LIN {X 0,Y 130.101,Z 635.486,A -85,B 0,C 180,E1 -28089.915,E2 -28089.915} C_VEL
LIN {X 0,Y 131.994,Z 639.477,A -85,B 0,C 180,E1 -28094.65,E2 -28094.65} C_VEL
LIN {X 0,Y 134.028,Z 643.617,A -85,B 0,C 180,E1 -28098.338,E2 -28098.338} C_VEL
LIN {X 0,Y 135.61,Z 647.254,A -85,B 0,C 180,E1 -28100.774,E2 -28100.774} C_VEL
LIN {X 0,Y 137.735,Z 654.472,A -85,B 0,C 180,E1 -28103.892,E2 -28103.892} C_VEL
LIN {X 0,Y 137.859,Z 654.961,A -85,B 0,C 180,E1 -28104.069,E2 -28104.069} C_VEL
LIN {X 0,Y 135.744,Z 673.421,A -85,B 0,C 180,E1 -28104.773,E2 -28104.773} C_VEL
LIN {X 0,Y 133.064,Z 685.971,A -85,B 0,C 180,E1 -28105.484,E2 -28105.484} C_VEL
LIN {X 0,Y 129.454,Z 697.536,A -85,B 0,C 180,E1 -28106.398,E2 -28106.398} C_VEL
LIN {X 0,Y 124.264,Z 710.187,A -85,B 0,C 180,E1 -28107.914,E2 -28107.914} C_VEL
LIN {X 0,Y 118.421,Z 721.436,A -85,B 0,C 180,E1 -28109.785,E2 -28109.785} C_VEL
LIN {X 0,Y 112.069,Z 731.569,A -85,B 0,C 180,E1 -28112.163,E2 -28112.163} C_VEL
LIN {X 0,Y 105.268,Z 740.708,A -85,B 0,C 180,E1 -28115.136,E2 -28115.136} C_VEL
LIN {X 0,Y 97.575,Z 749.621,A -85,B 0,C 180,E1 -28119.266,E2 -28119.266} C_VEL
LIN {X 0,Y 91.733,Z 755.687,A -85,B 0,C 180,E1 -28123.304,E2 -28123.304} C_VEL
LIN {X 0,Y 85.339,Z 761.645,A -85,B 0,C 180,E1 -28128.795,E2 -28128.795} C_VEL
LIN {X 0,Y 79.706,Z 766.355,A -85,B 0,C 180,E1 -28135.037,E2 -28135.037} C_VEL
LIN {X 0,Y 75.138,Z 769.96,A -85,B 0,C 180,E1 -28142.122,E2 -28142.122} C_VEL
LIN {X 0,Y 72.891,Z 771.823,A -85,B 0,C 180,E1 -28147.32,E2 -28147.32} C_VEL
LIN {X 0,Y 70.141,Z 774.222,A -85,B 0,C 180,E1 -28158.445,E2 -28158.445} C_VEL
LIN {X 0,Y 69.62,Z 774.834,A -85,B 0,C 180,E1 -28164.211,E2 -28164.211} C_VEL
LIN {X 0,Y 69.697,Z 775.05,A -85,B 0,C 180,E1 -28170.005,E2 -28170.005} C_VEL
LIN {X 0,Y 70.018,Z 774.825,A -85,B 0,C 180,E1 -28175.766,E2 -28175.766} C_VEL
LIN {X 0,Y 72.282,Z 773.204,A -85,B 0,C 180,E1 -28186.964,E2 -28186.964} C_VEL
LIN {X 0,Y 74.383,Z 771.8,A -85,B 0,C 180,E1 -28192.211,E2 -28192.211} C_VEL
LIN {X 0,Y 78.746,Z 768.868,A -85,B 0,C 180,E1 -28199.402,E2 -28199.402} C_VEL
LIN {X 0,Y 84.587,Z 764.915,A -85,B 0,C 180,E1 -28205.568,E2 -28205.568} C_VEL
LIN {X 0,Y 91.639,Z 759.801,A -85,B 0,C 180,E1 -28210.688,E2 -28210.688} C_VEL
LIN {X 0,Y 95.835,Z 756.939,A -85,B 0,C 180,E1 -28212.898,E2 -28212.898} C_VEL
LIN {X 0,Y 96.87,Z 757.298,A -85,B 0,C 180,E1 -28213.574,E2 -28213.574} C_VEL
LIN {X 0,Y 98.917,Z 759.037,A -85,B 0,C 180,E1 -28215.28,E2 -28215.28} C_VEL
LIN {X 0,Y 97.206,Z 757.454,A -85,B 0,C 180,E1 -28217.356,E2 -28217.356} C_VEL
LIN {X 0,Y 92.069,Z 751.92,A -85,B 0,C 180,E1 -28222.362,E2 -28222.362} C_VEL
LIN {X 0,Y 90.262,Z 751.095,A -85,B 0,C 180,E1 -28223.926,E2 -28223.926} C_VEL
LIN {X 0,Y 88.148,Z 750.795,A -85,B 0,C 180,E1 -28226.075,E2 -28226.075} C_VEL
LIN {X 0,Y 85.833,Z 749.445,A -85,B 0,C 180,E1 -28230.575,E2 -28230.575} C_VEL
LIN {X 0,Y 84.652,Z 747.487,A -85,B 0,C 180,E1 -28235.474,E2 -28235.474} C_VEL
LIN {X 0,Y 82.936,Z 746.489,A -85,B 0,C 180,E1 -28240.187,E2 -28240.187} C_VEL
LIN {X 0,Y 83.105,Z 742.849,A -85,B 0,C 180,E1 -28250.263,E2 -28250.263} C_VEL
LIN {X 0,Y 83.768,Z 741.308,A -85,B 0,C 180,E1 -28255.188,E2 -28255.188} C_VEL
LIN {X 0,Y 85.278,Z 739.422,A -85,B 0,C 180,E1 -28260,E2 -28260} C_VEL
LIN {X 0,Y 85.366,Z 739.328,A -85,B 0,C 180,E1 -28260.283,E2 -28260.283} C_VEL
LIN {X 0,Y 85.77,Z 738.947,A -85,B 0,C 180,E1 -28262.962,E2 -28262.962} C_VEL
LIN {X 0,Y 86.107,Z 739.875,A -85,B 0,C 180,E1 -28271.99,E2 -28271.99} C_VEL
LIN {X 0,Y 87.578,Z 739.192,A -85,B 0,C 180,E1 -28274.351,E2 -28274.351} C_VEL
LIN {X 0,Y 94.778,Z 735.064,A -85,B 0,C 180,E1 -28280.479,E2 -28280.479} C_VEL
LIN {X 0,Y 97.805,Z 733.364,A -85,B 0,C 180,E1 -28282.53,E2 -28282.53} C_VEL
LIN {X 0,Y 107.635,Z 727.025,A -85,B 0,C 180,E1 -28287.198,E2 -28287.198} C_VEL
LIN {X 0,Y 110.924,Z 724.845,A -85,B 0,C 180,E1 -28288.551,E2 -28288.551} C_VEL
LIN {X 0,Y 110.69,Z 725.783,A -85,B 0,C 180,E1 -28289.183,E2 -28289.183} C_VEL
LIN {X 0,Y 103.664,Z 735.37,A -85,B 0,C 180,E1 -28292.059,E2 -28292.059} C_VEL
LIN {X 0,Y 96.172,Z 744.056,A -85,B 0,C 180,E1 -28295.777,E2 -28295.777} C_VEL
LIN {X 0,Y 88.222,Z 751.991,A -85,B 0,C 180,E1 -28300.812,E2 -28300.812} C_VEL
LIN {X 0,Y 81.241,Z 757.929,A -85,B 0,C 180,E1 -28306.201,E2 -28306.201} C_VEL
LIN {X 0,Y 75.13,Z 762.615,A -85,B 0,C 180,E1 -28312.547,E2 -28312.547} C_VEL
LIN {X 0,Y 70.064,Z 766.192,A -85,B 0,C 180,E1 -28319.893,E2 -28319.893} C_VEL
LIN {X 0,Y 67.35,Z 768.037,A -85,B 0,C 180,E1 -28325.324,E2 -28325.324} C_VEL
LIN {X 0,Y 65.246,Z 769.422,A -85,B 0,C 180,E1 -28331.141,E2 -28331.141} C_VEL
LIN {X 0,Y 62.947,Z 771.009,A -85,B 0,C 180,E1 -28343.584,E2 -28343.584} C_VEL
LIN {X 0,Y 62.722,Z 771.232,A -85,B 0,C 180,E1 -28349.995,E2 -28349.995} C_VEL
LIN {X 0,Y 62.94,Z 771.037,A -85,B 0,C 180,E1 -28356.406,E2 -28356.406} C_VEL
LIN {X 0,Y 65.24,Z 769.487,A -85,B 0,C 180,E1 -28368.849,E2 -28368.849} C_VEL
LIN {X 0,Y 67.335,Z 768.13,A -85,B 0,C 180,E1 -28374.671,E2 -28374.671} C_VEL
LIN {X 0,Y 71.588,Z 765.258,A -85,B 0,C 180,E1 -28382.674,E2 -28382.674} C_VEL
LIN {X 0,Y 76.942,Z 761.361,A -85,B 0,C 180,E1 -28389.74,E2 -28389.74} C_VEL
LIN {X 0,Y 83.405,Z 756.331,A -85,B 0,C 180,E1 -28395.739,E2 -28395.739} C_VEL
LIN {X 0,Y 90.53,Z 749.996,A -85,B 0,C 180,E1 -28400.918,E2 -28400.918} C_VEL
LIN {X 0,Y 97.951,Z 742.366,A -85,B 0,C 180,E1 -28405.232,E2 -28405.232} C_VEL
LIN {X 0,Y 104.983,Z 733.989,A -85,B 0,C 180,E1 -28408.592,E2 -28408.592} C_VEL
LIN {X 0,Y 112.098,Z 724.12,A -85,B 0,C 180,E1 -28411.362,E2 -28411.362} C_VEL
LIN {X 0,Y 118.676,Z 713,A -85,B 0,C 180,E1 -28413.592,E2 -28413.592} C_VEL
LIN {X 0,Y 123.89,Z 702.094,A -85,B 0,C 180,E1 -28415.174,E2 -28415.174} C_VEL
LIN {X 0,Y 128.41,Z 690.022,A -85,B 0,C 180,E1 -28416.447,E2 -28416.447} C_VEL
LIN {X 0,Y 131.787,Z 677.536,A -85,B 0,C 180,E1 -28417.401,E2 -28417.401} C_VEL
LIN {X 0,Y 134.061,Z 664.506,A -85,B 0,C 180,E1 -28418.001,E2 -28418.001} C_VEL
LIN {X 0,Y 134.925,Z 656.287,A -85,B 0,C 180,E1 -28418.316,E2 -28418.316} C_VEL
LIN {X 0,Y 132.623,Z 650.593,A -85,B 0,C 180,E1 -28421.96,E2 -28421.96} C_VEL
LIN {X 0,Y 131.039,Z 647.12,A -85,B 0,C 180,E1 -28424.964,E2 -28424.964} C_VEL
LIN {X 0,Y 129.869,Z 644.563,A -85,B 0,C 180,E1 -28427.697,E2 -28427.697} C_VEL
LIN {X 0,Y 128.772,Z 641.834,A -85,B 0,C 180,E1 -28431.17,E2 -28431.17} C_VEL
LIN {X 0,Y 127.754,Z 638.206,A -85,B 0,C 180,E1 -28440,E2 -28440} C_VEL
LIN {X 0,Y 128.97,Z 642.374,A -85,B 0,C 180,E1 -28449.211,E2 -28449.211} C_VEL
LIN {X 0,Y 130.645,Z 646.219,A -85,B 0,C 180,E1 -28453.811,E2 -28453.811} C_VEL
LIN {X 0,Y 132.545,Z 650.383,A -85,B 0,C 180,E1 -28457.537,E2 -28457.537} C_VEL
LIN {X 0,Y 133.588,Z 653.255,A -85,B 0,C 180,E1 -28459.346,E2 -28459.346} C_VEL
LIN {X 0,Y 134.794,Z 657.852,A -85,B 0,C 180,E1 -28461.406,E2 -28461.406} C_VEL
LIN {X 0,Y 132.765,Z 674.133,A -85,B 0,C 180,E1 -28462.022,E2 -28462.022} C_VEL
LIN {X 0,Y 129.886,Z 686.836,A -85,B 0,C 180,E1 -28462.736,E2 -28462.736} C_VEL
LIN {X 0,Y 125.679,Z 699.334,A -85,B 0,C 180,E1 -28463.704,E2 -28463.704} C_VEL
LIN {X 0,Y 120.342,Z 711.571,A -85,B 0,C 180,E1 -28465.158,E2 -28465.158} C_VEL
LIN {X 0,Y 114.312,Z 722.477,A -85,B 0,C 180,E1 -28466.948,E2 -28466.948} C_VEL
LIN {X 0,Y 107.011,Z 733.323,A -85,B 0,C 180,E1 -28469.525,E2 -28469.525} C_VEL
LIN {X 0,Y 99.938,Z 742.137,A -85,B 0,C 180,E1 -28472.455,E2 -28472.455} C_VEL
LIN {X 0,Y 91.932,Z 750.729,A -85,B 0,C 180,E1 -28476.618,E2 -28476.618} C_VEL
LIN {X 0,Y 84.142,Z 757.985,A -85,B 0,C 180,E1 -28481.928,E2 -28481.928} C_VEL
LIN {X 0,Y 77.94,Z 763.129,A -85,B 0,C 180,E1 -28487.452,E2 -28487.452} C_VEL
LIN {X 0,Y 72.171,Z 767.458,A -85,B 0,C 180,E1 -28494.254,E2 -28494.254} C_VEL
LIN {X 0,Y 68.92,Z 769.755,A -85,B 0,C 180,E1 -28499.351,E2 -28499.351} C_VEL
LIN {X 0,Y 66.352,Z 771.617,A -85,B 0,C 180,E1 -28504.939,E2 -28504.939} C_VEL
LIN {X 0,Y 64.452,Z 773.016,A -85,B 0,C 180,E1 -28510.911,E2 -28510.911} C_VEL
LIN {X 0,Y 63.177,Z 774.017,A -85,B 0,C 180,E1 -28517.151,E2 -28517.151} C_VEL
LIN {X 0,Y 62.555,Z 774.629,A -85,B 0,C 180,E1 -28523.555,E2 -28523.555} C_VEL
LIN {X 0,Y 62.607,Z 774.846,A -85,B 0,C 180,E1 -28530.006,E2 -28530.006} C_VEL
LIN {X 0,Y 62.958,Z 774.62,A -85,B 0,C 180,E1 -28536.415,E2 -28536.415} C_VEL
LIN {X 0,Y 63.936,Z 774.004,A -85,B 0,C 180,E1 -28542.705,E2 -28542.705} C_VEL
LIN {X 0,Y 67.87,Z 771.594,A -85,B 0,C 180,E1 -28554.475,E2 -28554.475} C_VEL
LIN {X 0,Y 72.662,Z 768.663,A -85,B 0,C 180,E1 -28562.144,E2 -28562.144} C_VEL
LIN {X 0,Y 78.934,Z 764.71,A -85,B 0,C 180,E1 -28568.56,E2 -28568.56} C_VEL
LIN {X 0,Y 86.371,Z 759.609,A -85,B 0,C 180,E1 -28573.765,E2 -28573.765} C_VEL
LIN {X 0,Y 89.11,Z 757.647,A -85,B 0,C 180,E1 -28575.226,E2 -28575.226} C_VEL
LIN {X 0,Y 88.589,Z 756.273,A -85,B 0,C 180,E1 -28577.598,E2 -28577.598} C_VEL
LIN {X 0,Y 86.995,Z 755.555,A -85,B 0,C 180,E1 -28579.738,E2 -28579.738} C_VEL
LIN {X 0,Y 83.333,Z 754.787,A -85,B 0,C 180,E1 -28583.818,E2 -28583.818} C_VEL
LIN {X 0,Y 80.607,Z 753.671,A -85,B 0,C 180,E1 -28588.457,E2 -28588.457} C_VEL
LIN {X 0,Y 79.042,Z 752.041,A -85,B 0,C 180,E1 -28593.604,E2 -28593.604} C_VEL
LIN {X 0,Y 77.483,Z 750.845,A -85,B 0,C 180,E1 -28598.727,E2 -28598.727} C_VEL
LIN {X 0,Y 80.273,Z 743.799,A -85,B 0,C 180,E1 -28621.798,E2 -28621.798} C_VEL
LIN {X 0,Y 87.221,Z 739.406,A -85,B 0,C 180,E1 -28633.989,E2 -28633.989} C_VEL
LIN {X 0,Y 87.578,Z 739.192,A -85,B 0,C 180,E1 -28634.351,E2 -28634.351} C_VEL
LIN {X 0,Y 89.334,Z 738.402,A -85,B 0,C 180,E1 -28636.653,E2 -28636.653} C_VEL
LIN {X 0,Y 94.231,Z 737.919,A -85,B 0,C 180,E1 -28644.554,E2 -28644.554} C_VEL
LIN {X 0,Y 96.716,Z 736.808,A -85,B 0,C 180,E1 -28646.252,E2 -28646.252} C_VEL
LIN {X 0,Y 100.251,Z 734.753,A -85,B 0,C 180,E1 -28647.772,E2 -28647.772} C_VEL
LIN {X 0,Y 100.04,Z 735.616,A -85,B 0,C 180,E1 -28648.619,E2 -28648.619} C_VEL
LIN {X 0,Y 93.013,Z 743.428,A -85,B 0,C 180,E1 -28651.777,E2 -28651.777} C_VEL
LIN {X 0,Y 85.011,Z 751.089,A -85,B 0,C 180,E1 -28656.282,E2 -28656.282} C_VEL
LIN {X 0,Y 78.699,Z 756.328,A -85,B 0,C 180,E1 -28660.612,E2 -28660.612} C_VEL
LIN {X 0,Y 71.682,Z 761.409,A -85,B 0,C 180,E1 -28666.656,E2 -28666.656} C_VEL
LIN {X 0,Y 65.756,Z 765.341,A -85,B 0,C 180,E1 -28673.99,E2 -28673.99} C_VEL
LIN {X 0,Y 60.978,Z 768.243,A -85,B 0,C 180,E1 -28682.541,E2 -28682.541} C_VEL
LIN {X 0,Y 58.576,Z 769.627,A -85,B 0,C 180,E1 -28688.897,E2 -28688.897} C_VEL
LIN {X 0,Y 55.914,Z 771.214,A -85,B 0,C 180,E1 -28702.773,E2 -28702.773} C_VEL
LIN {X 0,Y 55.649,Z 771.436,A -85,B 0,C 180,E1 -28709.994,E2 -28709.994} C_VEL
LIN {X 0,Y 55.908,Z 771.241,A -85,B 0,C 180,E1 -28717.215,E2 -28717.215} C_VEL
LIN {X 0,Y 58.569,Z 769.691,A -85,B 0,C 180,E1 -28731.093,E2 -28731.093} C_VEL
LIN {X 0,Y 60.961,Z 768.334,A -85,B 0,C 180,E1 -28737.455,E2 -28737.455} C_VEL
LIN {X 0,Y 65.72,Z 765.462,A -85,B 0,C 180,E1 -28746.02,E2 -28746.02} C_VEL
LIN {X 0,Y 71.623,Z 761.565,A -85,B 0,C 180,E1 -28753.376,E2 -28753.376} C_VEL
LIN {X 0,Y 78.616,Z 756.535,A -85,B 0,C 180,E1 -28759.445,E2 -28759.445} C_VEL
LIN {X 0,Y 86.23,Z 750.198,A -85,B 0,C 180,E1 -28764.583,E2 -28764.583} C_VEL
LIN {X 0,Y 94.364,Z 742.272,A -85,B 0,C 180,E1 -28768.918,E2 -28768.918} C_VEL
LIN {X 0,Y 102.927,Z 732.412,A -85,B 0,C 180,E1 -28772.572,E2 -28772.572} C_VEL
LIN {X 0,Y 110.359,Z 722.044,A -85,B 0,C 180,E1 -28775.152,E2 -28775.152} C_VEL
LIN {X 0,Y 117.242,Z 710.355,A -85,B 0,C 180,E1 -28777.159,E2 -28777.159} C_VEL
LIN {X 0,Y 122.546,Z 698.849,A -85,B 0,C 180,E1 -28778.624,E2 -28778.624} C_VEL
LIN {X 0,Y 126.994,Z 686.168,A -85,B 0,C 180,E1 -28779.743,E2 -28779.743} C_VEL
LIN {X 0,Y 130.191,Z 673.179,A -85,B 0,C 180,E1 -28780.551,E2 -28780.551} C_VEL
LIN {X 0,Y 132.076,Z 659.981,A -85,B 0,C 180,E1 -28781.087,E2 -28781.087} C_VEL
LIN {X 0,Y 130.017,Z 654.538,A -85,B 0,C 180,E1 -28785.097,E2 -28785.097} C_VEL
LIN {X 0,Y 128.555,Z 651.086,A -85,B 0,C 180,E1 -28788.769,E2 -28788.769} C_VEL
LIN {X 0,Y 127.631,Z 648.65,A -85,B 0,C 180,E1 -28792.087,E2 -28792.087} C_VEL
LIN {X 0,Y 126.874,Z 645.374,A -85,B 0,C 180,E1 -28800,E2 -28800} C_VEL
LIN {X 0,Y 127.833,Z 649.157,A -85,B 0,C 180,E1 -28808.381,E2 -28808.381} C_VEL
LIN {X 0,Y 129.209,Z 652.691,A -85,B 0,C 180,E1 -28812.666,E2 -28812.666} C_VEL
LIN {X 0,Y 130.913,Z 656.84,A -85,B 0,C 180,E1 -28816.407,E2 -28816.407} C_VEL
LIN {X 0,Y 131.78,Z 659.784,A -85,B 0,C 180,E1 -28818.135,E2 -28818.135} C_VEL
LIN {X 0,Y 132.024,Z 660.831,A -85,B 0,C 180,E1 -28818.626,E2 -28818.626} C_VEL
LIN {X 0,Y 130.145,Z 674.683,A -85,B 0,C 180,E1 -28819.16,E2 -28819.16} C_VEL
LIN {X 0,Y 127.018,Z 687.602,A -85,B 0,C 180,E1 -28819.853,E2 -28819.853} C_VEL
LIN {X 0,Y 122.949,Z 699.261,A -85,B 0,C 180,E1 -28820.687,E2 -28820.687} C_VEL
LIN {X 0,Y 117.499,Z 711.372,A -85,B 0,C 180,E1 -28822.021,E2 -28822.021} C_VEL
LIN {X 0,Y 111.276,Z 722.276,A -85,B 0,C 180,E1 -28823.689,E2 -28823.689} C_VEL
LIN {X 0,Y 103.692,Z 733.121,A -85,B 0,C 180,E1 -28826.105,E2 -28826.105} C_VEL
LIN {X 0,Y 96.304,Z 741.934,A -85,B 0,C 180,E1 -28828.877,E2 -28828.877} C_VEL
LIN {X 0,Y 87.866,Z 750.526,A -85,B 0,C 180,E1 -28832.883,E2 -28832.883} C_VEL
LIN {X 0,Y 80.035,Z 757.41,A -85,B 0,C 180,E1 -28837.794,E2 -28837.794} C_VEL
LIN {X 0,Y 72.859,Z 762.925,A -85,B 0,C 180,E1 -28843.667,E2 -28843.667} C_VEL
LIN {X 0,Y 66.524,Z 767.254,A -85,B 0,C 180,E1 -28850.67,E2 -28850.67} C_VEL
LIN {X 0,Y 62.901,Z 769.551,A -85,B 0,C 180,E1 -28856.044,E2 -28856.044} C_VEL
LIN {X 0,Y 59.955,Z 771.412,A -85,B 0,C 180,E1 -28862.045,E2 -28862.045} C_VEL
LIN {X 0,Y 57.761,Z 772.811,A -85,B 0,C 180,E1 -28868.598,E2 -28868.598} C_VEL
LIN {X 0,Y 56.265,Z 773.812,A -85,B 0,C 180,E1 -28875.54,E2 -28875.54} C_VEL
LIN {X 0,Y 55.512,Z 774.425,A -85,B 0,C 180,E1 -28882.733,E2 -28882.733} C_VEL
LIN {X 0,Y 55.506,Z 774.641,A -85,B 0,C 180,E1 -28890.006,E2 -28890.006} C_VEL
LIN {X 0,Y 55.927,Z 774.416,A -85,B 0,C 180,E1 -28897.225,E2 -28897.225} C_VEL
LIN {X 0,Y 58.854,Z 772.794,A -85,B 0,C 180,E1 -28910.998,E2 -28910.998} C_VEL
LIN {X 0,Y 61.493,Z 771.39,A -85,B 0,C 180,E1 -28917.21,E2 -28917.21} C_VEL
LIN {X 0,Y 66.78,Z 768.458,A -85,B 0,C 180,E1 -28925.374,E2 -28925.374} C_VEL
LIN {X 0,Y 73.534,Z 764.505,A -85,B 0,C 180,E1 -28931.998,E2 -28931.998} C_VEL
LIN {X 0,Y 81.211,Z 759.537,A -85,B 0,C 180,E1 -28937.128,E2 -28937.128} C_VEL
LIN {X 0,Y 80.023,Z 758.768,A -85,B 0,C 180,E1 -28939.377,E2 -28939.377} C_VEL
LIN {X 0,Y 75.364,Z 757.491,A -85,B 0,C 180,E1 -28945.977,E2 -28945.977} C_VEL
LIN {X 0,Y 71.348,Z 752.029,A -85,B 0,C 180,E1 -28968.638,E2 -28968.638} C_VEL
LIN {X 0,Y 81.659,Z 744.392,A -85,B 0,C 180,E1 -28994.963,E2 -28994.963} C_VEL
LIN {X 0,Y 85.958,Z 742.211,A -85,B 0,C 180,E1 -28999.09,E2 -28999.09} C_VEL
LIN {X 0,Y 94.238,Z 738.135,A -85,B 0,C 180,E1 -29004.99,E2 -29004.99} C_VEL
LIN {X 0,Y 96.716,Z 736.808,A -85,B 0,C 180,E1 -29006.252,E2 -29006.252} C_VEL
LIN {X 0,Y 95.752,Z 737.763,A -85,B 0,C 180,E1 -29006.451,E2 -29006.451} C_VEL
LIN {X 0,Y 90.525,Z 741.419,A -85,B 0,C 180,E1 -29005.328,E2 -29005.328} C_VEL
LIN {X 0,Y 84.388,Z 745.051,A -85,B 0,C 180,E1 -29003.097,E2 -29003.097} C_VEL
LIN {X 0,Y 80.227,Z 747.13,A -85,B 0,C 180,E1 -29000.612,E2 -29000.612} C_VEL
LIN {X 0,Y 75.908,Z 748.925,A -85,B 0,C 180,E1 -28996.127,E2 -28996.127} C_VEL
LIN {X 0,Y 65.957,Z 754.628,A -85,B 0,C 180,E1 -28973.884,E2 -28973.884} C_VEL
LIN {X 0,Y 67.632,Z 759.85,A -85,B 0,C 180,E1 -28948.697,E2 -28948.697} C_VEL
LIN {X 0,Y 71.427,Z 761.31,A -85,B 0,C 180,E1 -28940.993,E2 -28940.993} C_VEL
LIN {X 0,Y 72.467,Z 761.915,A -85,B 0,C 180,E1 -28938.717,E2 -28938.717} C_VEL
LIN {X 0,Y 63.44,Z 767.03,A -85,B 0,C 180,E1 -28931.665,E2 -28931.665} C_VEL
LIN {X 0,Y 59.022,Z 769.319,A -85,B 0,C 180,E1 -28926.546,E2 -28926.546} C_VEL
LIN {X 0,Y 55.275,Z 771.184,A -85,B 0,C 180,E1 -28920.577,E2 -28920.577} C_VEL
LIN {X 0,Y 50.172,Z 773.594,A -85,B 0,C 180,E1 -28906.277,E2 -28906.277} C_VEL
LIN {X 0,Y 48.893,Z 774.211,A -85,B 0,C 180,E1 -28898.271,E2 -28898.271} C_VEL
LIN {X 0,Y 48.423,Z 774.437,A -85,B 0,C 180,E1 -28890.007,E2 -28890.007} C_VEL
LIN {X 0,Y 48.472,Z 774.22,A -85,B 0,C 180,E1 -28881.671,E2 -28881.671} C_VEL
LIN {X 0,Y 51.174,Z 772.605,A -85,B 0,C 180,E1 -28865.677,E2 -28865.677} C_VEL
LIN {X 0,Y 53.75,Z 771.206,A -85,B 0,C 180,E1 -28858.473,E2 -28858.473} C_VEL
LIN {X 0,Y 59.09,Z 768.271,A -85,B 0,C 180,E1 -28849.152,E2 -28849.152} C_VEL
LIN {X 0,Y 65.675,Z 764.305,A -85,B 0,C 180,E1 -28841.497,E2 -28841.497} C_VEL
LIN {X 0,Y 74.001,Z 758.608,A -85,B 0,C 180,E1 -28834.738,E2 -28834.738} C_VEL
LIN {X 0,Y 82.774,Z 751.559,A -85,B 0,C 180,E1 -28829.518,E2 -28829.518} C_VEL
LIN {X 0,Y 91.572,Z 743.304,A -85,B 0,C 180,E1 -28825.614,E2 -28825.614} C_VEL
LIN {X 0,Y 99.196,Z 734.858,A -85,B 0,C 180,E1 -28822.931,E2 -28822.931} C_VEL
LIN {X 0,Y 107.028,Z 724.426,A -85,B 0,C 180,E1 -28820.664,E2 -28820.664} C_VEL
LIN {X 0,Y 114.221,Z 712.682,A -85,B 0,C 180,E1 -28818.922,E2 -28818.922} C_VEL
LIN {X 0,Y 119.725,Z 701.262,A -85,B 0,C 180,E1 -28817.711,E2 -28817.711} C_VEL
LIN {X 0,Y 124.229,Z 689.153,A -85,B 0,C 180,E1 -28816.876,E2 -28816.876} C_VEL
LIN {X 0,Y 127.715,Z 675.876,A -85,B 0,C 180,E1 -28816.221,E2 -28816.221} C_VEL
LIN {X 0,Y 129.547,Z 664.049,A -85,B 0,C 180,E1 -28815.739,E2 -28815.739} C_VEL
LIN {X 0,Y 128.25,Z 660.288,A -85,B 0,C 180,E1 -28812.662,E2 -28812.662} C_VEL
LIN {X 0,Y 127.211,Z 657.494,A -85,B 0,C 180,E1 -28809.54,E2 -28809.54} C_VEL
LIN {X 0,Y 126.484,Z 655.285,A -85,B 0,C 180,E1 -28806.38,E2 -28806.38} C_VEL
LIN {X 0,Y 125.989,Z 652.577,A -85,B 0,C 180,E1 -28800,E2 -28800} C_VEL
LIN {X 0,Y 126.739,Z 655.984,A -85,B 0,C 180,E1 -28792.031,E2 -28792.031} C_VEL
LIN {X 0,Y 127.908,Z 659.378,A -85,B 0,C 180,E1 -28787.908,E2 -28787.908} C_VEL
LIN {X 0,Y 129.287,Z 663.248,A -85,B 0,C 180,E1 -28784.431,E2 -28784.431} C_VEL
LIN {X 0,Y 129.501,Z 663.935,A -85,B 0,C 180,E1 -28783.927,E2 -28783.927} C_VEL
LIN {X 0,Y 127.151,Z 677.322,A -85,B 0,C 180,E1 -28783.338,E2 -28783.338} C_VEL
LIN {X 0,Y 123.86,Z 689.18,A -85,B 0,C 180,E1 -28782.584,E2 -28782.584} C_VEL
LIN {X 0,Y 119.339,Z 700.928,A -85,B 0,C 180,E1 -28781.573,E2 -28781.573} C_VEL
LIN {X 0,Y 113.867,Z 711.978,A -85,B 0,C 180,E1 -28780.251,E2 -28780.251} C_VEL
LIN {X 0,Y 107.576,Z 722.245,A -85,B 0,C 180,E1 -28778.575,E2 -28778.575} C_VEL
LIN {X 0,Y 99.861,Z 732.613,A -85,B 0,C 180,E1 -28776.184,E2 -28776.184} C_VEL
LIN {X 0,Y 92.355,Z 740.997,A -85,B 0,C 180,E1 -28773.39,E2 -28773.39} C_VEL
LIN {X 0,Y 83.914,Z 749.02,A -85,B 0,C 180,E1 -28769.434,E2 -28769.434} C_VEL
LIN {X 0,Y 76.863,Z 754.757,A -85,B 0,C 180,E1 -28765.37,E2 -28765.37} C_VEL
LIN {X 0,Y 69.087,Z 760.203,A -85,B 0,C 180,E1 -28759.717,E2 -28759.717} C_VEL
LIN {X 0,Y 62.162,Z 764.467,A -85,B 0,C 180,E1 -28752.708,E2 -28752.708} C_VEL
LIN {X 0,Y 58.165,Z 766.722,A -85,B 0,C 180,E1 -28747.16,E2 -28747.16} C_VEL
LIN {X 0,Y 54.743,Z 768.539,A -85,B 0,C 180,E1 -28740.891,E2 -28740.891} C_VEL
LIN {X 0,Y 50.037,Z 770.861,A -85,B 0,C 180,E1 -28726.307,E2 -28726.307} C_VEL
LIN {X 0,Y 48.874,Z 771.445,A -85,B 0,C 180,E1 -28718.261,E2 -28718.261} C_VEL
LIN {X 0,Y 48.565,Z 771.64,A -85,B 0,C 180,E1 -28709.993,E2 -28709.993} C_VEL
LIN {X 0,Y 48.878,Z 771.418,A -85,B 0,C 180,E1 -28701.726,E2 -28701.726} C_VEL
LIN {X 0,Y 50.04,Z 770.816,A -85,B 0,C 180,E1 -28693.679,E2 -28693.679} C_VEL
LIN {X 0,Y 54.761,Z 768.448,A -85,B 0,C 180,E1 -28679.105,E2 -28679.105} C_VEL
LIN {X 0,Y 60.158,Z 765.547,A -85,B 0,C 180,E1 -28670.011,E2 -28670.011} C_VEL
LIN {X 0,Y 66.696,Z 761.615,A -85,B 0,C 180,E1 -28662.464,E2 -28662.464} C_VEL
LIN {X 0,Y 74.275,Z 756.534,A -85,B 0,C 180,E1 -28656.452,E2 -28656.452} C_VEL
LIN {X 0,Y 82.373,Z 750.135,A -85,B 0,C 180,E1 -28651.432,E2 -28651.432} C_VEL
LIN {X 0,Y 88.024,Z 745.015,A -85,B 0,C 180,E1 -28648.559,E2 -28648.559} C_VEL
LIN {X 0,Y 89.392,Z 743.169,A -85,B 0,C 180,E1 -28646.973,E2 -28646.973} C_VEL
LIN {X 0,Y 80.227,Z 747.13,A -85,B 0,C 180,E1 -28640.612,E2 -28640.612} C_VEL
LIN {X 0,Y 74.947,Z 749.727,A -85,B 0,C 180,E1 -28636.69,E2 -28636.69} C_VEL
LIN {X 0,Y 64.868,Z 754.966,A -85,B 0,C 180,E1 -28627.631,E2 -28627.631} C_VEL
LIN {X 0,Y 62.176,Z 756.388,A -85,B 0,C 180,E1 -28623.108,E2 -28623.108} C_VEL
LIN {X 0,Y 61.539,Z 756.762,A -85,B 0,C 180,E1 -28621.431,E2 -28621.431} C_VEL
LIN {X 0,Y 60.042,Z 761.988,A -85,B 0,C 180,E1 -28592.082,E2 -28592.082} C_VEL
LIN {X 0,Y 62.054,Z 763.068,A -85,B 0,C 180,E1 -28585.509,E2 -28585.509} C_VEL
LIN {X 0,Y 63.705,Z 764.094,A -85,B 0,C 180,E1 -28580.564,E2 -28580.564} C_VEL
LIN {X 0,Y 55.821,Z 768.048,A -85,B 0,C 180,E1 -28573.834,E2 -28573.834} C_VEL
LIN {X 0,Y 49.303,Z 770.979,A -85,B 0,C 180,E1 -28564.772,E2 -28564.772} C_VEL
LIN {X 0,Y 43.412,Z 773.389,A -85,B 0,C 180,E1 -28548.9,E2 -28548.9} C_VEL
LIN {X 0,Y 41.897,Z 774.006,A -85,B 0,C 180,E1 -28539.665,E2 -28539.665} C_VEL
LIN {X 0,Y 41.323,Z 774.232,A -85,B 0,C 180,E1 -28530.008,E2 -28530.008} C_VEL
LIN {X 0,Y 41.446,Z 774.015,A -85,B 0,C 180,E1 -28520.246,E2 -28520.246} C_VEL
LIN {X 0,Y 44.766,Z 772.4,A -85,B 0,C 180,E1 -28501.911,E2 -28501.911} C_VEL
LIN {X 0,Y 47.81,Z 771.001,A -85,B 0,C 180,E1 -28493.994,E2 -28493.994} C_VEL
LIN {X 0,Y 53.898,Z 768.067,A -85,B 0,C 180,E1 -28484.189,E2 -28484.189} C_VEL
LIN {X 0,Y 61.195,Z 764.102,A -85,B 0,C 180,E1 -28476.504,E2 -28476.504} C_VEL
LIN {X 0,Y 69.482,Z 758.893,A -85,B 0,C 180,E1 -28470.381,E2 -28470.381} C_VEL
LIN {X 0,Y 78.01,Z 752.593,A -85,B 0,C 180,E1 -28465.733,E2 -28465.733} C_VEL
LIN {X 0,Y 87.161,Z 744.591,A -85,B 0,C 180,E1 -28461.998,E2 -28461.998} C_VEL
LIN {X 0,Y 96.646,Z 734.656,A -85,B 0,C 180,E1 -28459.043,E2 -28459.043} C_VEL
LIN {X 0,Y 104.734,Z 724.225,A -85,B 0,C 180,E1 -28457.029,E2 -28457.029} C_VEL
LIN {X 0,Y 112.123,Z 712.482,A -85,B 0,C 180,E1 -28455.493,E2 -28455.493} C_VEL
LIN {X 0,Y 117.634,Z 701.359,A -85,B 0,C 180,E1 -28454.437,E2 -28454.437} C_VEL
LIN {X 0,Y 122.227,Z 689.37,A -85,B 0,C 180,E1 -28453.719,E2 -28453.719} C_VEL
LIN {X 0,Y 125.731,Z 676.524,A -85,B 0,C 180,E1 -28453.16,E2 -28453.16} C_VEL
LIN {X 0,Y 127.22,Z 668.095,A -85,B 0,C 180,E1 -28452.766,E2 -28452.766} C_VEL
LIN {X 0,Y 126.08,Z 664.34,A -85,B 0,C 180,E1 -28448.818,E2 -28448.818} C_VEL
LIN {X 0,Y 125.463,Z 662.101,A -85,B 0,C 180,E1 -28445.626,E2 -28445.626} C_VEL
LIN {X 0,Y 125.115,Z 659.699,A -85,B 0,C 180,E1 -28440,E2 -28440} C_VEL
LIN {X 0,Y 125.671,Z 662.859,A -85,B 0,C 180,E1 -28432.771,E2 -28432.771} C_VEL
LIN {X 0,Y 126.577,Z 666.11,A -85,B 0,C 180,E1 -28428.794,E2 -28428.794} C_VEL
LIN {X 0,Y 127.166,Z 668.141,A -85,B 0,C 180,E1 -28426.839,E2 -28426.839} C_VEL
LIN {X 0,Y 124.226,Z 681.703,A -85,B 0,C 180,E1 -28426.241,E2 -28426.241} C_VEL
LIN {X 0,Y 120.593,Z 693.091,A -85,B 0,C 180,E1 -28425.49,E2 -28425.49} C_VEL
LIN {X 0,Y 115.764,Z 704.452,A -85,B 0,C 180,E1 -28424.516,E2 -28424.516} C_VEL
LIN {X 0,Y 109.245,Z 716.295,A -85,B 0,C 180,E1 -28423.114,E2 -28423.114} C_VEL
LIN {X 0,Y 101.986,Z 726.856,A -85,B 0,C 180,E1 -28421.345,E2 -28421.345} C_VEL
LIN {X 0,Y 94.062,Z 736.369,A -85,B 0,C 180,E1 -28419.049,E2 -28419.049} C_VEL
LIN {X 0,Y 84.825,Z 745.508,A -85,B 0,C 180,E1 -28415.686,E2 -28415.686} C_VEL
LIN {X 0,Y 75.926,Z 752.852,A -85,B 0,C 180,E1 -28411.554,E2 -28411.554} C_VEL
LIN {X 0,Y 67.432,Z 758.74,A -85,B 0,C 180,E1 -28406.479,E2 -28406.479} C_VEL
LIN {X 0,Y 59.559,Z 763.386,A -85,B 0,C 180,E1 -28400.076,E2 -28400.076} C_VEL
LIN {X 0,Y 52.685,Z 766.925,A -85,B 0,C 180,E1 -28391.826,E2 -28391.826} C_VEL
LIN {X 0,Y 48.78,Z 768.743,A -85,B 0,C 180,E1 -28385.182,E2 -28385.182} C_VEL
LIN {X 0,Y 43.272,Z 771.065,A -85,B 0,C 180,E1 -28368.947,E2 -28368.947} C_VEL
LIN {X 0,Y 41.877,Z 771.649,A -85,B 0,C 180,E1 -28359.653,E2 -28359.653} C_VEL
LIN {X 0,Y 41.469,Z 771.845,A -85,B 0,C 180,E1 -28349.992,E2 -28349.992} C_VEL
LIN {X 0,Y 41.881,Z 771.623,A -85,B 0,C 180,E1 -28340.331,E2 -28340.331} C_VEL
LIN {X 0,Y 43.276,Z 771.021,A -85,B 0,C 180,E1 -28331.038,E2 -28331.038} C_VEL
LIN {X 0,Y 48.799,Z 768.654,A -85,B 0,C 180,E1 -28314.816,E2 -28314.816} C_VEL
LIN {X 0,Y 54.909,Z 765.753,A -85,B 0,C 180,E1 -28305.246,E2 -28305.246} C_VEL
LIN {X 0,Y 62.125,Z 761.82,A -85,B 0,C 180,E1 -28297.629,E2 -28297.629} C_VEL
LIN {X 0,Y 70.29,Z 756.74,A -85,B 0,C 180,E1 -28291.793,E2 -28291.793} C_VEL
LIN {X 0,Y 78.896,Z 750.342,A -85,B 0,C 180,E1 -28287.018,E2 -28287.018} C_VEL
LIN {X 0,Y 79.584,Z 749.578,A -85,B 0,C 180,E1 -28286.203,E2 -28286.203} C_VEL
LIN {X 0,Y 74.338,Z 751.551,A -85,B 0,C 180,E1 -28282.22,E2 -28282.22} C_VEL
LIN {X 0,Y 66.405,Z 754.444,A -85,B 0,C 180,E1 -28272.221,E2 -28272.221} C_VEL
LIN {X 0,Y 61.539,Z 756.762,A -85,B 0,C 180,E1 -28261.431,E2 -28261.431} C_VEL
LIN {X 0,Y 59.506,Z 758.118,A -85,B 0,C 180,E1 -28256.326,E2 -28256.326} C_VEL
LIN {X 0,Y 55.587,Z 760.943,A -85,B 0,C 180,E1 -28247.669,E2 -28247.669} C_VEL
LIN {X 0,Y 53.092,Z 763.498,A -85,B 0,C 180,E1 -28237.93,E2 -28237.93} C_VEL
LIN {X 0,Y 53.408,Z 764.536,A -85,B 0,C 180,E1 -28231.706,E2 -28231.706} C_VEL
LIN {X 0,Y 54.898,Z 765.293,A -85,B 0,C 180,E1 -28226.049,E2 -28226.049} C_VEL
LIN {X 0,Y 55.039,Z 766.026,A -85,B 0,C 180,E1 -28222.828,E2 -28222.828} C_VEL
LIN {X 0,Y 48.366,Z 768.909,A -85,B 0,C 180,E1 -28216.607,E2 -28216.607} C_VEL
LIN {X 0,Y 43.673,Z 770.774,A -85,B 0,C 180,E1 -28210.078,E2 -28210.078} C_VEL
LIN {X 0,Y 36.787,Z 773.184,A -85,B 0,C 180,E1 -28192.473,E2 -28192.473} C_VEL
LIN {X 0,Y 34.929,Z 773.802,A -85,B 0,C 180,E1 -28181.618,E2 -28181.618} C_VEL
LIN {X 0,Y 34.237,Z 774.028,A -85,B 0,C 180,E1 -28170.01,E2 -28170.01} C_VEL
LIN {X 0,Y 34.467,Z 773.81,A -85,B 0,C 180,E1 -28158.245,E2 -28158.245} C_VEL
LIN {X 0,Y 38.622,Z 772.195,A -85,B 0,C 180,E1 -28136.925,E2 -28136.925} C_VEL
LIN {X 0,Y 42.245,Z 770.796,A -85,B 0,C 180,E1 -28128.294,E2 -28128.294} C_VEL
LIN {X 0,Y 49.196,Z 767.862,A -85,B 0,C 180,E1 -28118.226,E2 -28118.226} C_VEL
LIN {X 0,Y 57.252,Z 763.898,A -85,B 0,C 180,E1 -28110.776,E2 -28110.776} C_VEL
LIN {X 0,Y 66.413,Z 758.536,A -85,B 0,C 180,E1 -28104.934,E2 -28104.934} C_VEL
LIN {X 0,Y 76.762,Z 751.152,A -85,B 0,C 180,E1 -28100.222,E2 -28100.222} C_VEL
LIN {X 0,Y 86.379,Z 742.899,A -85,B 0,C 180,E1 -28097.073,E2 -28097.073} C_VEL
LIN {X 0,Y 94.563,Z 734.453,A -85,B 0,C 180,E1 -28094.962,E2 -28094.962} C_VEL
LIN {X 0,Y 102.882,Z 724.025,A -85,B 0,C 180,E1 -28093.253,E2 -28093.253} C_VEL
LIN {X 0,Y 110.441,Z 712.283,A -85,B 0,C 180,E1 -28091.948,E2 -28091.948} C_VEL
LIN {X 0,Y 116.583,Z 699.964,A -85,B 0,C 180,E1 -28090.98,E2 -28090.98} C_VEL
LIN {X 0,Y 121.448,Z 687.012,A -85,B 0,C 180,E1 -28090.357,E2 -28090.357} C_VEL
LIN {X 0,Y 124.711,Z 674.513,A -85,B 0,C 180,E1 -28089.898,E2 -28089.898} C_VEL
LIN {X 0,Y 125.046,Z 672.664,A -85,B 0,C 180,E1 -28089.819,E2 -28089.819} C_VEL
LIN {X 0,Y 124.402,Z 669.185,A -85,B 0,C 180,E1 -28085.47,E2 -28085.47} C_VEL
LIN {X 0,Y 124.144,Z 666.888,A -85,B 0,C 180,E1 -28080,E2 -28080} C_VEL
LIN {X 0,Y 124.403,Z 669.681,A -85,B 0,C 180,E1 -28073.512,E2 -28073.512} C_VEL
LIN {X 0,Y 124.94,Z 672.55,A -85,B 0,C 180,E1 -28069.924,E2 -28069.924} C_VEL
LIN {X 0,Y 122.297,Z 683.479,A -85,B 0,C 180,E1 -28069.384,E2 -28069.384} C_VEL
LIN {X 0,Y 118.015,Z 695.853,A -85,B 0,C 180,E1 -28068.643,E2 -28068.643} C_VEL
LIN {X 0,Y 113.239,Z 706.297,A -85,B 0,C 180,E1 -28067.806,E2 -28067.806} C_VEL
LIN {X 0,Y 106.573,Z 717.783,A -85,B 0,C 180,E1 -28066.565,E2 -28066.565} C_VEL
LIN {X 0,Y 99.122,Z 728.123,A -85,B 0,C 180,E1 -28065.012,E2 -28065.012} C_VEL
LIN {X 0,Y 91.766,Z 736.571,A -85,B 0,C 180,E1 -28063.186,E2 -28063.186} C_VEL
LIN {X 0,Y 82.158,Z 745.711,A -85,B 0,C 180,E1 -28060.202,E2 -28060.202} C_VEL
LIN {X 0,Y 72.804,Z 753.056,A -85,B 0,C 180,E1 -28056.488,E2 -28056.488} C_VEL
LIN {X 0,Y 63.79,Z 758.943,A -85,B 0,C 180,E1 -28051.798,E2 -28051.798} C_VEL
LIN {X 0,Y 55.273,Z 763.589,A -85,B 0,C 180,E1 -28045.727,E2 -28045.727} C_VEL
LIN {X 0,Y 47.636,Z 767.129,A -85,B 0,C 180,E1 -28037.522,E2 -28037.522} C_VEL
LIN {X 0,Y 43.172,Z 768.947,A -85,B 0,C 180,E1 -28030.619,E2 -28030.619} C_VEL
LIN {X 0,Y 36.624,Z 771.27,A -85,B 0,C 180,E1 -28012.558,E2 -28012.558} C_VEL
LIN {X 0,Y 34.894,Z 771.854,A -85,B 0,C 180,E1 -28001.609,E2 -28001.609} C_VEL
LIN {X 0,Y 34.391,Z 772.049,A -85,B 0,C 180,E1 -27989.99,E2 -27989.99} C_VEL
LIN {X 0,Y 34.898,Z 771.828,A -85,B 0,C 180,E1 -27978.372,E2 -27978.372} C_VEL
LIN {X 0,Y 39.454,Z 770.242,A -85,B 0,C 180,E1 -27957.687,E2 -27957.687} C_VEL
LIN {X 0,Y 43.191,Z 768.859,A -85,B 0,C 180,E1 -27949.382,E2 -27949.382} C_VEL
LIN {X 0,Y 50.119,Z 765.958,A -85,B 0,C 180,E1 -27939.524,E2 -27939.524} C_VEL
LIN {X 0,Y 58.067,Z 762.026,A -85,B 0,C 180,E1 -27932.078,E2 -27932.078} C_VEL
LIN {X 0,Y 66.454,Z 757.176,A -85,B 0,C 180,E1 -27926.814,E2 -27926.814} C_VEL
LIN {X 0,Y 68.428,Z 755.492,A -85,B 0,C 180,E1 -27924.257,E2 -27924.257} C_VEL
LIN {X 0,Y 52.813,Z 761.703,A -85,B 0,C 180,E1 -27892.353,E2 -27892.353} C_VEL
LIN {X 0,Y 53.408,Z 764.536,A -85,B 0,C 180,E1 -27871.706,E2 -27871.706} C_VEL
LIN {X 0,Y 53.146,Z 765.119,A -85,B 0,C 180,E1 -27869.336,E2 -27869.336} C_VEL
LIN {X 0,Y 51.503,Z 766.167,A -85,B 0,C 180,E1 -27866.765,E2 -27866.765} C_VEL
LIN {X 0,Y 47.991,Z 767.669,A -85,B 0,C 180,E1 -27863.869,E2 -27863.869} C_VEL
LIN {X 0,Y 39.894,Z 770.184,A -85,B 0,C 180,E1 -27858.291,E2 -27858.291} C_VEL
LIN {X 0,Y 37.552,Z 770.85,A -85,B 0,C 180,E1 -27855.349,E2 -27855.349} C_VEL
LIN {X 0,Y 30.355,Z 772.98,A -85,B 0,C 180,E1 -27837.597,E2 -27837.597} C_VEL
LIN {X 0,Y 28.011,Z 773.597,A -85,B 0,C 180,E1 -27824.544,E2 -27824.544} C_VEL
LIN {X 0,Y 27.123,Z 773.823,A -85,B 0,C 180,E1 -27810.013,E2 -27810.013} C_VEL
LIN {X 0,Y 27.537,Z 773.605,A -85,B 0,C 180,E1 -27795.226,E2 -27795.226} C_VEL
LIN {X 0,Y 32.885,Z 771.99,A -85,B 0,C 180,E1 -27770.137,E2 -27770.137} C_VEL
LIN {X 0,Y 37.222,Z 770.591,A -85,B 0,C 180,E1 -27760.968,E2 -27760.968} C_VEL
LIN {X 0,Y 45.135,Z 767.657,A -85,B 0,C 180,E1 -27751.099,E2 -27751.099} C_VEL
LIN {X 0,Y 53.96,Z 763.694,A -85,B 0,C 180,E1 -27744.273,E2 -27744.273} C_VEL
LIN {X 0,Y 63.342,Z 758.57,A -85,B 0,C 180,E1 -27739.297,E2 -27739.297} C_VEL
LIN {X 0,Y 72.955,Z 752.185,A -85,B 0,C 180,E1 -27735.584,E2 -27735.584} C_VEL
LIN {X 0,Y 82.893,Z 744.186,A -85,B 0,C 180,E1 -27732.855,E2 -27732.855} C_VEL
LIN {X 0,Y 92.981,Z 734.251,A -85,B 0,C 180,E1 -27730.722,E2 -27730.722} C_VEL
LIN {X 0,Y 101.489,Z 723.824,A -85,B 0,C 180,E1 -27729.346,E2 -27729.346} C_VEL
LIN {X 0,Y 109.194,Z 712.083,A -85,B 0,C 180,E1 -27728.307,E2 -27728.307} C_VEL
LIN {X 0,Y 115.216,Z 700.289,A -85,B 0,C 180,E1 -27727.548,E2 -27727.548} C_VEL
LIN {X 0,Y 120.376,Z 686.816,A -85,B 0,C 180,E1 -27727.037,E2 -27727.037} C_VEL
LIN {X 0,Y 122.972,Z 677.344,A -85,B 0,C 180,E1 -27726.676,E2 -27726.676} C_VEL
LIN {X 0,Y 122.791,Z 675.512,A -85,B 0,C 180,E1 -27723.692,E2 -27723.692} C_VEL
LIN {X 0,Y 122.837,Z 674.015,A -85,B 0,C 180,E1 -27720,E2 -27720} C_VEL
LIN {X 0,Y 122.801,Z 676.432,A -85,B 0,C 180,E1 -27714.252,E2 -27714.252} C_VEL
LIN {X 0,Y 122.869,Z 677.362,A -85,B 0,C 180,E1 -27712.96,E2 -27712.96} C_VEL
LIN {X 0,Y 119.078,Z 690.212,A -85,B 0,C 180,E1 -27712.358,E2 -27712.358} C_VEL
LIN {X 0,Y 114.215,Z 701.93,A -85,B 0,C 180,E1 -27711.695,E2 -27711.695} C_VEL
LIN {X 0,Y 108.545,Z 712.578,A -85,B 0,C 180,E1 -27710.871,E2 -27710.871} C_VEL
LIN {X 0,Y 100.904,Z 724.017,A -85,B 0,C 180,E1 -27709.654,E2 -27709.654} C_VEL
LIN {X 0,Y 93.319,Z 733.218,A -85,B 0,C 180,E1 -27708.23,E2 -27708.23} C_VEL
LIN {X 0,Y 84.976,Z 741.604,A -85,B 0,C 180,E1 -27706.338,E2 -27706.338} C_VEL
LIN {X 0,Y 75.557,Z 749.475,A -85,B 0,C 180,E1 -27703.571,E2 -27703.571} C_VEL
LIN {X 0,Y 67.083,Z 755.367,A -85,B 0,C 180,E1 -27700.526,E2 -27700.526} C_VEL
LIN {X 0,Y 57.658,Z 760.813,A -85,B 0,C 180,E1 -27696.075,E2 -27696.075} C_VEL
LIN {X 0,Y 48.674,Z 765.08,A -85,B 0,C 180,E1 -27690.02,E2 -27690.02} C_VEL
LIN {X 0,Y 43.153,Z 767.333,A -85,B 0,C 180,E1 -27684.505,E2 -27684.505} C_VEL
LIN {X 0,Y 38.07,Z 769.151,A -85,B 0,C 180,E1 -27677.584,E2 -27677.584} C_VEL
LIN {X 0,Y 30.197,Z 771.474,A -85,B 0,C 180,E1 -27657.728,E2 -27657.728} C_VEL
LIN {X 0,Y 27.971,Z 772.058,A -85,B 0,C 180,E1 -27644.539,E2 -27644.539} C_VEL
LIN {X 0,Y 27.295,Z 772.254,A -85,B 0,C 180,E1 -27629.987,E2 -27629.987} C_VEL
LIN {X 0,Y 27.976,Z 772.033,A -85,B 0,C 180,E1 -27615.438,E2 -27615.438} C_VEL
LIN {X 0,Y 30.203,Z 771.431,A -85,B 0,C 180,E1 -27602.252,E2 -27602.252} C_VEL
LIN {X 0,Y 38.089,Z 769.065,A -85,B 0,C 180,E1 -27582.42,E2 -27582.42} C_VEL
LIN {X 0,Y 45.915,Z 766.164,A -85,B 0,C 180,E1 -27572.651,E2 -27572.651} C_VEL
LIN {X 0,Y 56.596,Z 761.223,A -85,B 0,C 180,E1 -27564.614,E2 -27564.614} C_VEL
LIN {X 0,Y 58.488,Z 760.064,A -85,B 0,C 180,E1 -27562.443,E2 -27562.443} C_VEL
LIN {X 0,Y 45.561,Z 765.653,A -85,B 0,C 180,E1 -27522.031,E2 -27522.031} C_VEL
LIN {X 0,Y 46.343,Z 766.621,A -85,B 0,C 180,E1 -27512.703,E2 -27512.703} C_VEL
LIN {X 0,Y 46.285,Z 767.774,A -85,B 0,C 180,E1 -27505.655,E2 -27505.655} C_VEL
LIN {X 0,Y 37.552,Z 770.85,A -85,B 0,C 180,E1 -27495.349,E2 -27495.349} C_VEL
LIN {X 0,Y 33.339,Z 771.99,A -85,B 0,C 180,E1 -27488.843,E2 -27488.843} C_VEL
LIN {X 0,Y 26.091,Z 773.183,A -85,B 0,C 180,E1 -27475.875,E2 -27475.875} C_VEL
LIN {X 0,Y 21.471,Z 773.568,A -85,B 0,C 180,E1 -27460.055,E2 -27460.055} C_VEL
LIN {X 0,Y 20.041,Z 773.578,A -85,B 0,C 180,E1 -27443.991,E2 -27443.991} C_VEL
LIN {X 0,Y 20.144,Z 773.492,A -85,B 0,C 180,E1 -27438.324,E2 -27438.324} C_VEL
LIN {X 0,Y 23.507,Z 772.786,A -85,B 0,C 180,E1 -27413.295,E2 -27413.295} C_VEL
LIN {X 0,Y 27.787,Z 771.785,A -85,B 0,C 180,E1 -27400.663,E2 -27400.663} C_VEL
LIN {X 0,Y 32.987,Z 770.386,A -85,B 0,C 180,E1 -27391.568,E2 -27391.568} C_VEL
LIN {X 0,Y 41.9,Z 767.453,A -85,B 0,C 180,E1 -27382.724,E2 -27382.724} C_VEL
LIN {X 0,Y 51.445,Z 763.49,A -85,B 0,C 180,E1 -27377.03,E2 -27377.03} C_VEL
LIN {X 0,Y 62.978,Z 757.404,A -85,B 0,C 180,E1 -27372.492,E2 -27372.492} C_VEL
LIN {X 0,Y 73.069,Z 750.745,A -85,B 0,C 180,E1 -27369.672,E2 -27369.672} C_VEL
LIN {X 0,Y 83.317,Z 742.493,A -85,B 0,C 180,E1 -27367.668,E2 -27367.668} C_VEL
LIN {X 0,Y 91.923,Z 734.049,A -85,B 0,C 180,E1 -27366.362,E2 -27366.362} C_VEL
LIN {X 0,Y 100.581,Z 723.623,A -85,B 0,C 180,E1 -27365.355,E2 -27365.355} C_VEL
LIN {X 0,Y 108.397,Z 711.883,A -85,B 0,C 180,E1 -27364.598,E2 -27364.598} C_VEL
LIN {X 0,Y 114.196,Z 700.784,A -85,B 0,C 180,E1 -27364.052,E2 -27364.052} C_VEL
LIN {X 0,Y 119.239,Z 688.034,A -85,B 0,C 180,E1 -27363.69,E2 -27363.69} C_VEL
LIN {X 0,Y 120.985,Z 682.385,A -85,B 0,C 180,E1 -27363.517,E2 -27363.517} C_VEL
LIN {X 0,Y 121.088,Z 681.034,A -85,B 0,C 180,E1 -27360,E2 -27360} C_VEL
LIN {X 0,Y 120.896,Z 682.437,A -85,B 0,C 180,E1 -27356.112,E2 -27356.112} C_VEL
LIN {X 0,Y 116.608,Z 694.931,A -85,B 0,C 180,E1 -27355.578,E2 -27355.578} C_VEL
LIN {X 0,Y 111.111,Z 706.695,A -85,B 0,C 180,E1 -27354.973,E2 -27354.973} C_VEL
LIN {X 0,Y 104.194,Z 718.184,A -85,B 0,C 180,E1 -27354.174,E2 -27354.174} C_VEL
LIN {X 0,Y 96.429,Z 728.526,A -85,B 0,C 180,E1 -27353.194,E2 -27353.194} C_VEL
LIN {X 0,Y 88.708,Z 736.974,A -85,B 0,C 180,E1 -27351.992,E2 -27351.992} C_VEL
LIN {X 0,Y 78.489,Z 746.117,A -85,B 0,C 180,E1 -27350.019,E2 -27350.019} C_VEL
LIN {X 0,Y 68.39,Z 753.461,A -85,B 0,C 180,E1 -27347.464,E2 -27347.464} C_VEL
LIN {X 0,Y 58.442,Z 759.349,A -85,B 0,C 180,E1 -27344.141,E2 -27344.141} C_VEL
LIN {X 0,Y 48.7,Z 763.997,A -85,B 0,C 180,E1 -27339.703,E2 -27339.703} C_VEL
LIN {X 0,Y 39.453,Z 767.537,A -85,B 0,C 180,E1 -27332.939,E2 -27332.939} C_VEL
LIN {X 0,Y 33.688,Z 769.355,A -85,B 0,C 180,E1 -27326.541,E2 -27326.541} C_VEL
LIN {X 0,Y 24.152,Z 771.678,A -85,B 0,C 180,E1 -27305.572,E2 -27305.572} C_VEL
LIN {X 0,Y 21.182,Z 772.263,A -85,B 0,C 180,E1 -27289.36,E2 -27289.36} C_VEL
LIN {X 0,Y 20.214,Z 772.458,A -85,B 0,C 180,E1 -27269.983,E2 -27269.983} C_VEL
LIN {X 0,Y 24.16,Z 771.635,A -85,B 0,C 180,E1 -27234.406,E2 -27234.406} C_VEL
LIN {X 0,Y 33.708,Z 769.27,A -85,B 0,C 180,E1 -27213.471,E2 -27213.471} C_VEL
LIN {X 0,Y 42.501,Z 766.37,A -85,B 0,C 180,E1 -27204.547,E2 -27204.547} C_VEL
LIN {X 0,Y 45.575,Z 765.156,A -85,B 0,C 180,E1 -27202.277,E2 -27202.277} C_VEL
LIN {X 0,Y 47.957,Z 764.037,A -85,B 0,C 180,E1 -27199.068,E2 -27199.068} C_VEL
LIN {X 0,Y 39.435,Z 768.464,A -85,B 0,C 180,E1 -27153.027,E2 -27153.027} C_VEL
LIN {X 0,Y 34.071,Z 770.364,A -85,B 0,C 180,E1 -27145.617,E2 -27145.617} C_VEL
LIN {X 0,Y 24.286,Z 772.775,A -85,B 0,C 180,E1 -27125.382,E2 -27125.382} C_VEL
LIN {X 0,Y 21.22,Z 773.392,A -85,B 0,C 180,E1 -27109.359,E2 -27109.359} C_VEL
LIN {X 0,Y 20.016,Z 773.618,A -85,B 0,C 180,E1 -27090.017,E2 -27090.017} C_VEL
LIN {X 0,Y 20.144,Z 773.492,A -85,B 0,C 180,E1 -27078.324,E2 -27078.324} C_VEL
LIN {X 0,Y 20.699,Z 773.325,A -85,B 0,C 180,E1 -27067.392,E2 -27067.392} C_VEL
LIN {X 0,Y 22.506,Z 772.585,A -85,B 0,C 180,E1 -27046.938,E2 -27046.938} C_VEL
LIN {X 0,Y 28.512,Z 770.641,A -85,B 0,C 180,E1 -27023.835,E2 -27023.835} C_VEL
LIN {X 0,Y 33.125,Z 769.293,A -85,B 0,C 180,E1 -27017.346,E2 -27017.346} C_VEL
LIN {X 0,Y 34.862,Z 768.752,A -85,B 0,C 180,E1 -27015.984,E2 -27015.984} C_VEL
LIN {X 0,Y 46.42,Z 764.719,A -85,B 0,C 180,E1 -27010.276,E2 -27010.276} C_VEL
LIN {X 0,Y 57.007,Z 759.825,A -85,B 0,C 180,E1 -27007.081,E2 -27007.081} C_VEL
LIN {X 0,Y 68.74,Z 752.929,A -85,B 0,C 180,E1 -27004.627,E2 -27004.627} C_VEL
LIN {X 0,Y 79.18,Z 745.265,A -85,B 0,C 180,E1 -27003.182,E2 -27003.182} C_VEL
LIN {X 0,Y 89.659,Z 735.637,A -85,B 0,C 180,E1 -27002.082,E2 -27002.082} C_VEL
LIN {X 0,Y 98.415,Z 725.712,A -85,B 0,C 180,E1 -27001.414,E2 -27001.414} C_VEL
LIN {X 0,Y 106.306,Z 714.537,A -85,B 0,C 180,E1 -27000.928,E2 -27000.928} C_VEL
LIN {X 0,Y 113.146,Z 702.173,A -85,B 0,C 180,E1 -27000.52,E2 -27000.52} C_VEL
LIN {X 0,Y 118.123,Z 690.396,A -85,B 0,C 180,E1 -27000.316,E2 -27000.316} C_VEL
LIN {X 0,Y 118.665,Z 688.811,A -85,B 0,C 180,E1 -27000.296,E2 -27000.296} C_VEL
LIN {X 0,Y 118.955,Z 687.931,A -85,B 0,C 180,E1 -27000,E2 -27000} C_VEL
LIN {X 0,Y 118.931,Z 687.987,A -85,B 0,C 180,E1 -26999.571,E2 -26999.571} C_VEL
LIN {X 0,Y 118.397,Z 689.568,A -85,B 0,C 180,E1 -26999.241,E2 -26999.241} C_VEL
LIN {X 0,Y 113.164,Z 702.08,A -85,B 0,C 180,E1 -26998.845,E2 -26998.845} C_VEL
LIN {X 0,Y 107.214,Z 712.976,A -85,B 0,C 180,E1 -26998.358,E2 -26998.358} C_VEL
LIN {X 0,Y 99.342,Z 724.419,A -85,B 0,C 180,E1 -26997.725,E2 -26997.725} C_VEL
LIN {X 0,Y 91.485,Z 733.622,A -85,B 0,C 180,E1 -26996.968,E2 -26996.968} C_VEL
LIN {X 0,Y 81.043,Z 743.488,A -85,B 0,C 180,E1 -26995.703,E2 -26995.703} C_VEL
LIN {X 0,Y 70.663,Z 751.414,A -85,B 0,C 180,E1 -26993.984,E2 -26993.984} C_VEL
LIN {X 0,Y 60.341,Z 757.753,A -85,B 0,C 180,E1 -26991.849,E2 -26991.849} C_VEL
LIN {X 0,Y 50.101,Z 762.785,A -85,B 0,C 180,E1 -26989.053,E2 -26989.053} C_VEL
LIN {X 0,Y 40.046,Z 766.687,A -85,B 0,C 180,E1 -26984.816,E2 -26984.816} C_VEL
LIN {X 0,Y 30.351,Z 769.56,A -85,B 0,C 180,E1 -26977.825,E2 -26977.825} C_VEL
LIN {X 0,Y 18.833,Z 771.882,A -85,B 0,C 180,E1 -26958.247,E2 -26958.247} C_VEL
LIN {X 0,Y 14.692,Z 772.467,A -85,B 0,C 180,E1 -26938.551,E2 -26938.551} C_VEL
LIN {X 0,Y 13.126,Z 772.662,A -85,B 0,C 180,E1 -26909.974,E2 -26909.974} C_VEL
LIN {X 0,Y 14.699,Z 772.442,A -85,B 0,C 180,E1 -26881.41,E2 -26881.41} C_VEL
LIN {X 0,Y 18.842,Z 771.841,A -85,B 0,C 180,E1 -26861.73,E2 -26861.73} C_VEL
LIN {X 0,Y 30.369,Z 769.476,A -85,B 0,C 180,E1 -26842.201,E2 -26842.201} C_VEL
LIN {X 0,Y 36.797,Z 767.631,A -85,B 0,C 180,E1 -26837.228,E2 -26837.228} C_VEL
LIN {X 0,Y 36.355,Z 767.585,A -85,B 0,C 180,E1 -26831.147,E2 -26831.147} C_VEL
LIN {X 0,Y 32.018,Z 769.223,A -85,B 0,C 180,E1 -26807.321,E2 -26807.321} C_VEL
LIN {X 0,Y 30.583,Z 770.156,A -85,B 0,C 180,E1 -26796.838,E2 -26796.838} C_VEL
LIN {X 0,Y 18.955,Z 772.57,A -85,B 0,C 180,E1 -26777.889,E2 -26777.889} C_VEL
LIN {X 0,Y 14.727,Z 773.188,A -85,B 0,C 180,E1 -26758.531,E2 -26758.531} C_VEL
LIN {X 0,Y 12.923,Z 773.413,A -85,B 0,C 180,E1 -26730.027,E2 -26730.027} C_VEL
LIN {X 0,Y 14.247,Z 773.195,A -85,B 0,C 180,E1 -26700.471,E2 -26700.471} C_VEL
LIN {X 0,Y 23.755,Z 771.579,A -85,B 0,C 180,E1 -26667.466,E2 -26667.466} C_VEL
LIN {X 0,Y 29.879,Z 770.181,A -85,B 0,C 180,E1 -26659.838,E2 -26659.838} C_VEL
LIN {X 0,Y 34.862,Z 768.752,A -85,B 0,C 180,E1 -26655.984,E2 -26655.984} C_VEL
LIN {X 0,Y 39.945,Z 767.125,A -85,B 0,C 180,E1 -26652.073,E2 -26652.073} C_VEL
LIN {X 0,Y 47.851,Z 763.93,A -85,B 0,C 180,E1 -26645.403,E2 -26645.403} C_VEL
LIN {X 0,Y 55.926,Z 760.017,A -85,B 0,C 180,E1 -26640.666,E2 -26640.666} C_VEL
LIN {X 0,Y 61.015,Z 757.263,A -85,B 0,C 180,E1 -26639.436,E2 -26639.436} C_VEL
LIN {X 0,Y 63.254,Z 755.977,A -85,B 0,C 180,E1 -26639.066,E2 -26639.066} C_VEL
LIN {X 0,Y 51.474,Z 762.006,A -85,B 0,C 180,E1 -26637.576,E2 -26637.576} C_VEL
LIN {X 0,Y 38.793,Z 766.891,A -85,B 0,C 180,E1 -26635.03,E2 -26635.03} C_VEL
LIN {X 0,Y 28.439,Z 769.765,A -85,B 0,C 180,E1 -26631.225,E2 -26631.225} C_VEL
LIN {X 0,Y 15.069,Z 772.087,A -85,B 0,C 180,E1 -26618.806,E2 -26618.806} C_VEL
LIN {X 0,Y 9.115,Z 772.671,A -85,B 0,C 180,E1 -26600.387,E2 -26600.387} C_VEL
LIN {X 0,Y 6.027,Z 772.867,A -85,B 0,C 180,E1 -26549.943,E2 -26549.943} C_VEL
LIN {X 0,Y 9.125,Z 772.647,A -85,B 0,C 180,E1 -26499.569,E2 -26499.569} C_VEL
LIN {X 0,Y 15.081,Z 772.045,A -85,B 0,C 180,E1 -26481.181,E2 -26481.181} C_VEL
LIN {X 0,Y 25.71,Z 770.267,A -85,B 0,C 180,E1 -26470.287,E2 -26470.287} C_VEL
LIN {X 0,Y 27.508,Z 769.889,A -85,B 0,C 180,E1 -26467.256,E2 -26467.256} C_VEL
LIN {X 0,Y 25.488,Z 770.466,A -85,B 0,C 180,E1 -26454.026,E2 -26454.026} C_VEL
LIN {X 0,Y 23.791,Z 770.979,A -85,B 0,C 180,E1 -26447.425,E2 -26447.425} C_VEL
LIN {X 0,Y 15.147,Z 772.365,A -85,B 0,C 180,E1 -26438.178,E2 -26438.178} C_VEL
LIN {X 0,Y 9.159,Z 772.984,A -85,B 0,C 180,E1 -26420.174,E2 -26420.174} C_VEL
LIN {X 0,Y 5.817,Z 773.208,A -85,B 0,C 180,E1 -26370.059,E2 -26370.059} C_VEL
LIN {X 0,Y 8.789,Z 772.991,A -85,B 0,C 180,E1 -26316.973,E2 -26316.973} C_VEL
LIN {X 0,Y 21.419,Z 771.373,A -85,B 0,C 180,E1 -26290.246,E2 -26290.246} C_VEL
LIN {X 0,Y 32.907,Z 768.734,A -85,B 0,C 180,E1 -26284.443,E2 -26284.443} C_VEL
LIN {X 0,Y 42.188,Z 765.82,A -85,B 0,C 180,E1 -26282.035,E2 -26282.035} C_VEL
LIN {X 0,Y 53.666,Z 761.049,A -85,B 0,C 180,E1 -26280.246,E2 -26280.246} C_VEL
LIN {X 0,Y 61.015,Z 757.263,A -85,B 0,C 180,E1 -26279.436,E2 -26279.436} C_VEL
LIN {X 0,Y 61.015,Z 757.263,A -85,B 0,C 180,E1 -26279.436,E2 -26279.436}

QRS_NEXT_CUT()

QRS_NEXT()
QRS_HOME()

END
